(* IEC 61131-3 sources: Industry-PLC-LLM/data/PLCBEAD_repo/PLCBEAD_PLCEmbed-main/PLC-BEAD/Source/GEB/FF_RSE, 1 file *)

(* ---- FF_RSE.ST ---- *)
FUNCTION_BLOCK FF_RSE
	VAR_INPUT
		CS :	BOOL;
		CR :	BOOL;
		RST :	BOOL;
	END_VAR

	VAR_OUTPUT
		Q :	BOOL;
	END_VAR

	VAR
		es :	BOOL;
		er :	BOOL;
	END_VAR

	IF RST THEN
		(* asynchronous reset *)
		Q := FALSE;
	ELSIF CR AND NOT er THEN
		(* rising edge on CR *)
		Q := FALSE;
	ELSIF CS AND NOT es THEN
		(* rising edge on CS *)
		Q := TRUE;
	END_IF;

	es := CS;
	er := CR;
END_FUNCTION_BLOCK

PROGRAM program0
  VAR
	CS  :	BOOL;
	CR  :	BOOL;
	RST :	BOOL;

	Q :	BOOL;

	func_block : FF_RSE;
  END_VAR
	func_block.CS  :=CS ;
	func_block.CR  :=CR ;
	func_block.RST :=RST;
	func_block();
	Q := func_block.Q;
END_PROGRAM
